TYPE ST_sample :
STRUCT
	title : STRING;
	id : UINT;
	datetime : DT;
END_STRUCT
END_TYPE

(* stored: Version 1.1.0.1, ProductVersion 3.1.4024.12
   DUT ST_Sample: Id {bc2e2569-3ce1-46e8-aebe-d9481538272a} *)
